// TIA Portal V18 export
// export: Created 2026-06-11T17:45:26.4811721Z, ExportSetting WithDefaults, DisplayName Totally Integrated Automation Portal, DisplayVersion V18, DisplayName TIA Portal Openness, DisplayVersion V18, DisplayName TIA Portal Version Control Interface, DisplayVersion V18, DisplayName STEP 7 Professional, DisplayVersion V18, DisplayName STEP 7 Safety, DisplayVersion V18, DisplayName WinCC Professional, DisplayVersion V18
Screen "Screen_2"  1920x1080, Number=2
  ScreenLayer 
    GraphicView "Graphic view_1" at 0,0 size 1920x1080  Picture=scadabai2_2
    IOField "I/O field_1" at 217,281 size 128x40  DataFormat=Decimal, FormatPattern=999.9, Mode=InOutput
      ProcessValue := AI_LT3203_PV
    IOField "I/O field_2" at 789,300 size 119x36  DataFormat=Decimal, FormatPattern=999.9, Mode=InOutput
      ProcessValue := AI_LT3209_PV
    IOField "I/O field_4" at 1252,490 size 121x36  DataFormat=Decimal, FormatPattern=99.9, Mode=InOutput
      ProcessValue := AI_TT3214_PV
    IOField "I/O field_5" at 1243,300 size 119x37  DataFormat=Decimal, FormatPattern=999.9, Mode=InOutput
      ProcessValue := AI_LT3213_PV
    IOField "I/O field_6" at 787,483 size 123x41  DataFormat=Decimal, FormatPattern=99.9, Mode=InOutput
      ProcessValue := AI_TT3208_PV
    IOField "I/O field_7" at 1715,304 size 116x37  DataFormat=Decimal, FormatPattern=999.9, Mode=InOutput
      ProcessValue := AI_LT3218_PV
    IOField "I/O field_3" at 216,492 size 125x36  DataFormat=Decimal, FormatPattern=99.9, Mode=InOutput
      ProcessValue := AI_TT3204_PV
    IOField "I/O field_8" at 1715,486 size 116x33  DataFormat=Decimal, FormatPattern=99.9, Mode=InOutput
      ProcessValue := AI_TT3219_PV
    Button "Button_1" at 13,612 size 150x45  Mode=Text, TextOff="CIP BON 1", TextOn="Text"
    Button "Button_2" at 23,948 size 148x79  Mode=Text, TextOff="CANH BAO", TextOn="Text"
    Button "Button_3" at 508,604 size 147x46  Mode=Text, TextOff="CIP BON CHUA 2", TextOn="Text"
    Button "Button_4" at 614,791 size 195x51  Mode=Text, TextOff="CIP BON CHUA", TextOn="Text"
    Button "Button_5" at 178,950 size 156x77  Mode=Text, TextOff="PLC", TextOn="Text"
    Button "Button_6" at 339,949 size 155x75  Mode=Text, TextOff="DO THI", TextOn="Text"
    Button "Button_7" at 505,949 size 144x76  Mode=Text, TextOff="THONG SO SAN PHAM", TextOn="Text"
    Button "Button_8" at 669,947 size 153x79  Mode=Text, TextOff="CHU TRINH", TextOn="Text"
    Button "Button_9" at 1018,606 size 150x47  Mode=Text, TextOff="CIP BON CHUA 3", TextOn="Text"
    Button "Button_10" at 724,703 size 198x67  Mode=Text, TextOff="MIXING CIP", TextOn="Text"
    Button "Button_11" at 943,723 size 180x108  Mode=Text, TextOff="CIP CONTROL SEQUENCE", TextOn="Text"
    Button "Button_12" at 1508,598 size 144x53  Mode=Text, TextOff="CIP BON CHUA 4", TextOn="Text"
    GraphicView "Graphic view_2" at 215,175 size 79x67  Picture=6a021ba1-5713-4731-bd8c-8271e17dea45
    GraphicView "Graphic view_3" at 644,649 size 79x71  Picture=6a021ba1-5713-4731-bd8c-8271e17dea45
    GraphicView "Graphic view_4" at 1212,173 size 79x70  Picture=6a021ba1-5713-4731-bd8c-8271e17dea45
    GraphicView "Graphic view_5" at 1695,176 size 80x68  Picture=6a021ba1-5713-4731-bd8c-8271e17dea45
    GraphicView "Graphic view_6" at 1634,530 size 79x71  Picture=6a021ba1-5713-4731-bd8c-8271e17dea45
    GraphicView "Graphic view_8" at 1632,648 size 78x74  Picture=6a021ba1-5713-4731-bd8c-8271e17dea45
    GraphicView "Graphic view_9" at 145,649 size 74x71  Picture=6a021ba1-5713-4731-bd8c-8271e17dea45
    GraphicView "Graphic view_10" at 1154,532 size 75x67  Picture=6a021ba1-5713-4731-bd8c-8271e17dea45
    GraphicView "Graphic view_11" at 1150,649 size 80x73  Picture=6a021ba1-5713-4731-bd8c-8271e17dea45
    GraphicView "Graphic view_12" at 648,533 size 76x68  Picture=6a021ba1-5713-4731-bd8c-8271e17dea45
    GraphicView "Graphic view_13" at 647,531 size 78x74  Picture=6a021ba1-5713-4731-bd8c-8271e17dea45
    GraphicView "Graphic view_14" at 140,531 size 84x71  Picture=6a021ba1-5713-4731-bd8c-8271e17dea45
    GraphicView "Graphic view_15" at 1268,572 size 63x77  Picture=cbacbd3b-9325-4287-a974-7519f4b351b9
    GraphicView "Graphic view_16" at 1268,572 size 67x78  Picture=cbacbd3b-9325-4287-a974-7519f4b351b9
    GraphicView "Graphic view_17" at 1729,575 size 67x73  Picture=cbacbd3b-9325-4287-a974-7519f4b351b9
    GraphicView "Graphic view_18" at 765,572 size 72x80  Picture=cbacbd3b-9325-4287-a974-7519f4b351b9
    Button "Button_13" at 845,949 size 131x72  Mode=Text, TextOff="NGUONG ANALOG", TextOn="Text"
    Button "Button_14" at 1000,951 size 144x73  Mode=Text, TextOff="PID", TextOn="Text"
    Button "Button_15" at 1173,948 size 154x75  Mode=Text, TextOff="DANG NHAP", TextOn="Text"
    Button "Button_16" at 1344,948 size 153x74  Mode=Text, TextOff="TAB OFF", TextOn="Text"
    Button "Button_17" at 1516,950 size 142x70  Mode=Text, TextOff="ASK", TextOn="Text"
    Button "Button_18" at 1681,849 size 111x76  Mode=Text, TextOff="MAN HINH", TextOn="Text"
    Button "Button_19" at 1628,793 size 183x48  Mode=Text, TextOff="CIP BON CHUA", TextOn="Text"
    GraphicView "Graphic view_7" at 60,132 size 1770x25  Picture=Graphic_16
    GraphicView "Graphic view_23" at 1705,132 size 37x41  Picture=Graphic_18
    GraphicView "Graphic view_29" at 1791,612 size 43x51  Picture=Graphic_20
    GraphicView "Graphic view_35" at 1652,594 size 40x64  Picture=Graphic_22
    GraphicView "Graphic view_48" at 1689,615 size 45x27  Picture=Graphic_23
    GraphicView "Graphic view_55" at 1651,491 size 21x44  Picture=Graphic_17
    GraphicView "Graphic view_67" at 1714,239 size 23x46  Picture=Graphic_17
    GraphicView "Graphic view_68" at 110,237 size 129x142  Picture=79334f88-f72e-4c6e-8b6a-52b316a98d43
    GraphicView "Graphic view_69" at 614,239 size 126x133  Picture=79334f88-f72e-4c6e-8b6a-52b316a98d43
    GraphicView "Graphic view_70" at 1117,240 size 115x136  Picture=79334f88-f72e-4c6e-8b6a-52b316a98d43
    GraphicView "Graphic view_71" at 1593,239 size 124x143  Picture=79334f88-f72e-4c6e-8b6a-52b316a98d43
    GraphicView "Graphic view_72" at 294,789 size 73x69  Picture=Graphic_25
    GraphicView "Graphic view_73" at 678,589 size 36x42  Picture=Graphic_25
    GraphicView "Graphic view_19" at 711,176 size 79x67  Picture=6a021ba1-5713-4731-bd8c-8271e17dea45
    GraphicView "Graphic view_20" at 264,573 size 72x80  Picture=cbacbd3b-9325-4287-a974-7519f4b351b9
    TextField "Text_field_Unit_I/O field_1" at 353,281 size 60x40  StyleItem=Text field, Text="<body><p>L</p></body>"
    TextField "Text_field_Unit_I/O field_2" at 916,300 size 60x36  StyleItem=Text field, Text="<body><p>L</p></body>"
    TextField "Text_field_Unit_I/O field_4" at 1381,490 size 60x36  StyleItem=Text field, Text="<body><p>°C</p></body>"
    TextField "Text_field_Unit_I/O field_5" at 1370,300 size 60x37  StyleItem=Text field, Text="<body><p>L</p></body>"
    TextField "Text_field_Unit_I/O field_6" at 918,483 size 60x41  StyleItem=Text field, Text="<body><p>°C</p></body>"
    TextField "Text_field_Unit_I/O field_7" at 1839,304 size 60x37  StyleItem=Text field, Text="<body><p>L</p></body>"
    TextField "Text_field_Unit_I/O field_3" at 349,492 size 60x36  StyleItem=Text field, Text="<body><p>°C</p></body>"
    TextField "Text_field_Unit_I/O field_8" at 1839,486 size 60x33  StyleItem=Text field, Text="<body><p>°C</p></body>"
